PROGRAM MAIN_Task1
VAR
    MachineSettingsServer : T_MachineSettingsServer; // Sends settings and loaded status to MachineSettingsClient running in separate context (task)
    Init            : BOOL := TRUE;

END_VAR

IF Init THEN
    // Manually resize the args buffer, as resizing 10,000 times produces a very long scan...
    Notifications.MachineSettingsUpdated.Args.Init(StreamLength := 60000);

    // Link the handler to the notification...
    Notifications.MachineSettingsLoaded
        .ClearNotificationHandlers()
    	.AddNotificationHandler(MAIN_Task2.MachineSettingsClient.OnSettingsLoaded);

    Notifications.MachineSettingsUpdated
        .ClearNotificationHandlers()
    	.AddNotificationHandler(MAIN_Task2.MachineSettingsClient.OnSettingsUpdated);

    Init := FALSE;
END_IF

// Run the server...
MachineSettingsServer.CyclicUpdate();

END_PROGRAM

(* stored: Version 1.1.0.1, ProductVersion 3.1.4024.12
   POU MAIN_Task1: Id {3afae642-2c54-4c29-a9d8-58ae31c6c9fc}, SpecialFunc None *)
